// TIA Portal V19 export
DATA_BLOCK "PSF DB"   // DB8
{ S7_Optimized_Access := 'TRUE' }
// stored: MemoryReserve 100
   VAR
      "PSF TANK" : Int;
   END_VAR
BEGIN
END_DATA_BLOCK
